SUBAPPLICATION Uebung_020c (* DigitalInput_I1 auf DigitalOutput_Q1; E_TON; Einschaltverzögert *)
  (* Standard: 61499-2; Description: Copyright (c) 2023 Meisterschulen am Ostbahnhof This program and the accompanying materials are made available under the terms of the Eclipse Public License 2.0 which is available at https://www.eclipse.org/legal/epl-2.0/ SPDX-License-Identifier: EPL-2.0 *)
  (* Version 1.0, 2023-10-23, Franz Höpfinger, Meisterschulen am Ostbahnhof *)
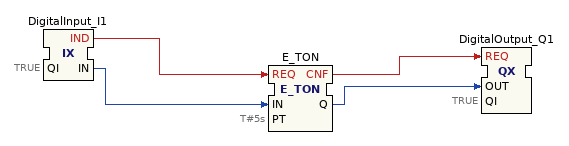
  FBS
    DigitalOutput_Q1 : QX(QI := TRUE);
    DigitalInput_I1 : IX(QI := TRUE);
    E_TON : E_TON(PT := T#5s);
  END_FBS
  EVENT_CONNECTIONS
    DigitalInput_I1.IND TO E_TON.REQ;
    E_TON.CNF TO DigitalOutput_Q1.REQ;
  END_CONNECTIONS
  DATA_CONNECTIONS
    DigitalInput_I1.IN TO E_TON.IN;
    E_TON.Q TO DigitalOutput_Q1.OUT;
  END_CONNECTIONS
END_SUBAPPLICATION
